// LS Electric XG5000 project: 2VFD2PUMPS
// PLC LSPLC

PROGRAM ECODELI (task: Scan Program)

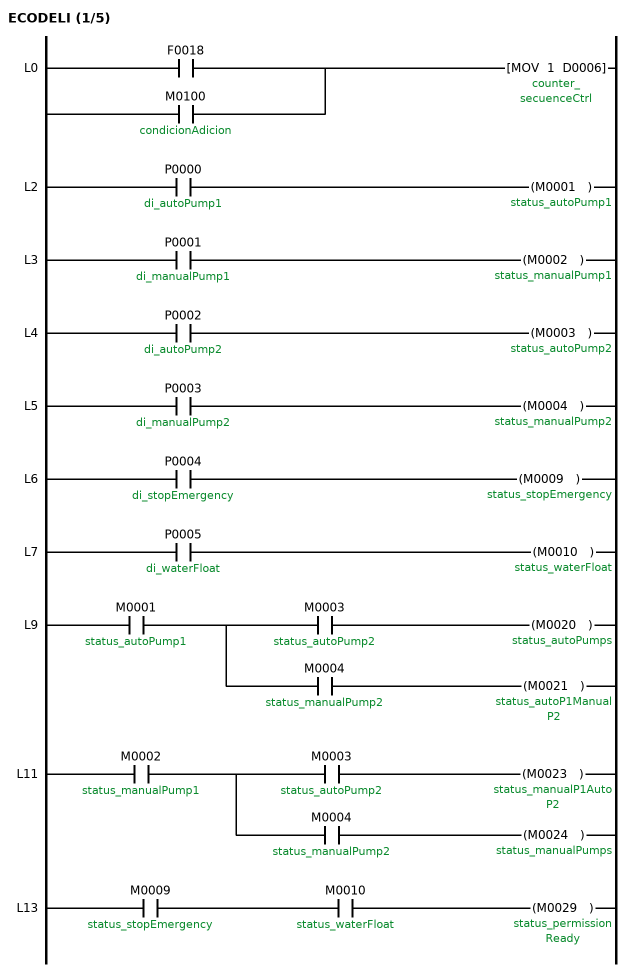
; L0
LOAD      F0018
OR        M0100	// condicionAdicion
MOV       1 D0006	// counter_secuenceCtrl
; L2
LOAD      P0000	// di_autoPump1
OUT       M0001	// status_autoPump1
; L3
LOAD      P0001	// di_manualPump1
OUT       M0002	// status_manualPump1
; L4
LOAD      P0002	// di_autoPump2
OUT       M0003	// status_autoPump2
; L5
LOAD      P0003	// di_manualPump2
OUT       M0004	// status_manualPump2
; L6
LOAD      P0004	// di_stopEmergency
OUT       M0009	// status_stopEmergency
; L7
LOAD      P0005	// di_waterFloat
OUT       M0010	// status_waterFloat
; L9
LOAD      M0001	// status_autoPump1
MPUSH
AND       M0003	// status_autoPump2
OUT       M0020	// status_autoPumps
MPOP
AND       M0004	// status_manualPump2
OUT       M0021	// status_autoP1ManualP2
; L11
LOAD      M0002	// status_manualPump1
MPUSH
AND       M0003	// status_autoPump2
OUT       M0023	// status_manualP1AutoP2
MPOP
AND       M0004	// status_manualPump2
OUT       M0024	// status_manualPumps
; L13
LOAD      M0009	// status_stopEmergency
AND       M0010	// status_waterFloat
OUT       M0029	// status_permissionReady

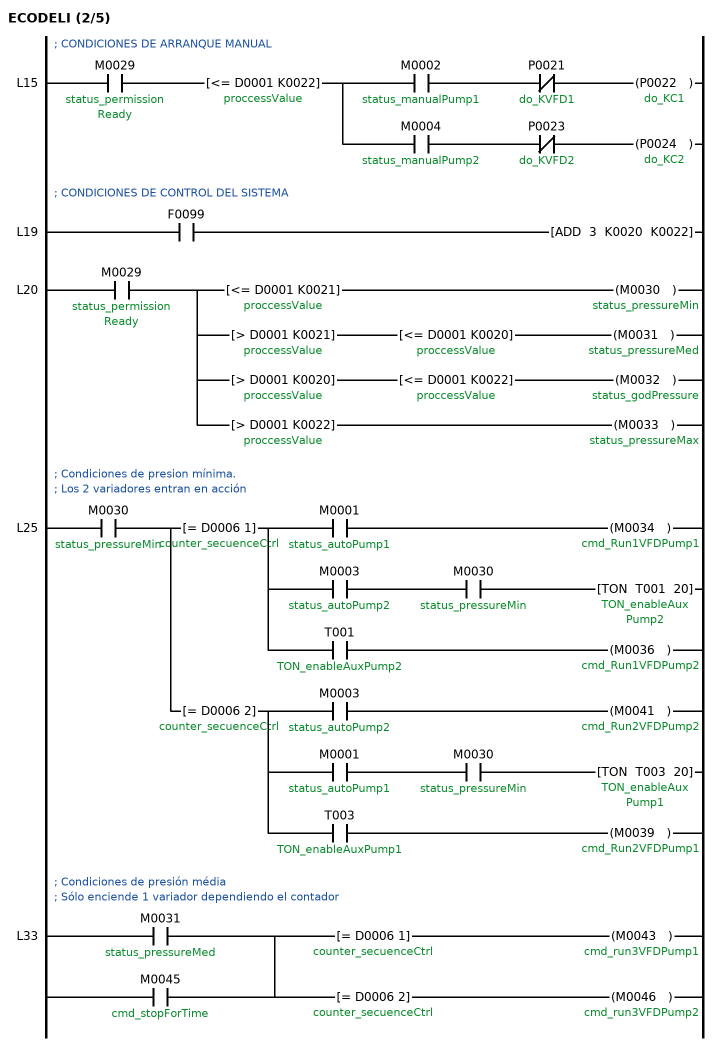
// CONDICIONES DE ARRANQUE MANUAL
; L15
LOAD      M0029	// status_permissionReady
AND<=     D0001 K0022	// proccessValue
MPUSH
AND       M0002	// status_manualPump1
AND NOT   P0021	// do_KVFD1
OUT       P0022	// do_KC1
MPOP
AND       M0004	// status_manualPump2
AND NOT   P0023	// do_KVFD2
OUT       P0024	// do_KC2
// CONDICIONES DE CONTROL DEL SISTEMA
; L19
LOAD      F0099
ADD       3 K0020 K0022
; L20
LOAD      M0029	// status_permissionReady
MPUSH
AND<=     D0001 K0021	// proccessValue
OUT       M0030	// status_pressureMin
MLOAD
AND>      D0001 K0021	// proccessValue
AND<=     D0001 K0020	// proccessValue
OUT       M0031	// status_pressureMed
MLOAD
AND>      D0001 K0020	// proccessValue
AND<=     D0001 K0022	// proccessValue
OUT       M0032	// status_godPressure
MPOP
AND>      D0001 K0022	// proccessValue
OUT       M0033	// status_pressureMax
// Condiciones de presion mínima.
// Los 2 variadores entran en acción
; L25
LOAD      M0030	// status_pressureMin
MPUSH
AND=      D0006 1	// counter_secuenceCtrl
MPUSH
AND       M0001	// status_autoPump1
OUT       M0034	// cmd_Run1VFDPump1
MLOAD
AND       M0003	// status_autoPump2
AND       M0030	// status_pressureMin
TON       T001 20	// TON_enableAuxPump2
MPOP
AND       T001	// TON_enableAuxPump2
OUT       M0036	// cmd_Run1VFDPump2
MPOP
AND=      D0006 2	// counter_secuenceCtrl
MPUSH
AND       M0003	// status_autoPump2
OUT       M0041	// cmd_Run2VFDPump2
MLOAD
AND       M0001	// status_autoPump1
AND       M0030	// status_pressureMin
TON       T003 20	// TON_enableAuxPump1
MPOP
AND       T003	// TON_enableAuxPump1
OUT       M0039	// cmd_Run2VFDPump1
// Condiciones de presión média
// Sólo enciende 1 variador dependiendo el contador
; L33
LOAD      M0031	// status_pressureMed
OR        M0045	// cmd_stopForTime
MPUSH
AND=      D0006 1	// counter_secuenceCtrl
OUT       M0043	// cmd_run3VFDPump1
MPOP
AND=      D0006 2	// counter_secuenceCtrl
OUT       M0046	// cmd_run3VFDPump2

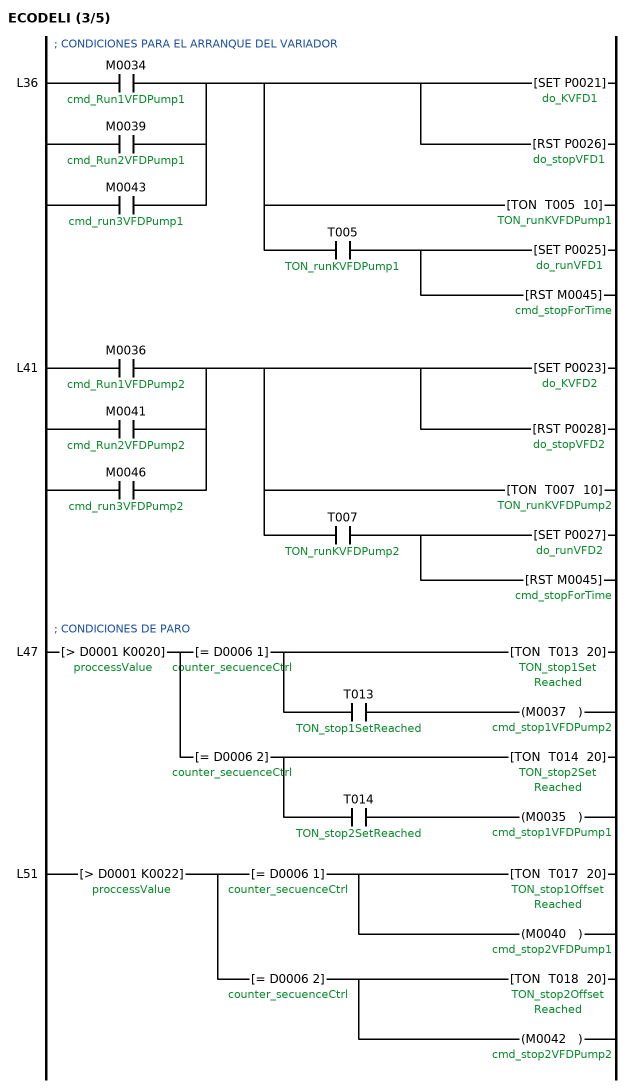
// CONDICIONES PARA EL ARRANQUE DEL VARIADOR
; L36
LOAD      M0034	// cmd_Run1VFDPump1
OR        M0039	// cmd_Run2VFDPump1
OR        M0043	// cmd_run3VFDPump1
SET       P0021	// do_KVFD1
RST       P0026	// do_stopVFD1
TON       T005 10	// TON_runKVFDPump1
AND       T005	// TON_runKVFDPump1
SET       P0025	// do_runVFD1
RST       M0045	// cmd_stopForTime
; L41
LOAD      M0036	// cmd_Run1VFDPump2
OR        M0041	// cmd_Run2VFDPump2
OR        M0046	// cmd_run3VFDPump2
SET       P0023	// do_KVFD2
RST       P0028	// do_stopVFD2
TON       T007 10	// TON_runKVFDPump2
AND       T007	// TON_runKVFDPump2
SET       P0027	// do_runVFD2
RST       M0045	// cmd_stopForTime
// CONDICIONES DE PARO
; L47
LOAD>     D0001 K0020	// proccessValue
MPUSH
AND=      D0006 1	// counter_secuenceCtrl
TON       T013 20	// TON_stop1SetReached
AND       T013	// TON_stop1SetReached
OUT       M0037	// cmd_stop1VFDPump2
MPOP
AND=      D0006 2	// counter_secuenceCtrl
TON       T014 20	// TON_stop2SetReached
AND       T014	// TON_stop2SetReached
OUT       M0035	// cmd_stop1VFDPump1
; L51
LOAD>     D0001 K0022	// proccessValue
MPUSH
AND=      D0006 1	// counter_secuenceCtrl
TON       T017 20	// TON_stop1OffsetReached
OUT       M0040	// cmd_stop2VFDPump1
MPOP
AND=      D0006 2	// counter_secuenceCtrl
TON       T018 20	// TON_stop2OffsetReached
OUT       M0042	// cmd_stop2VFDPump2

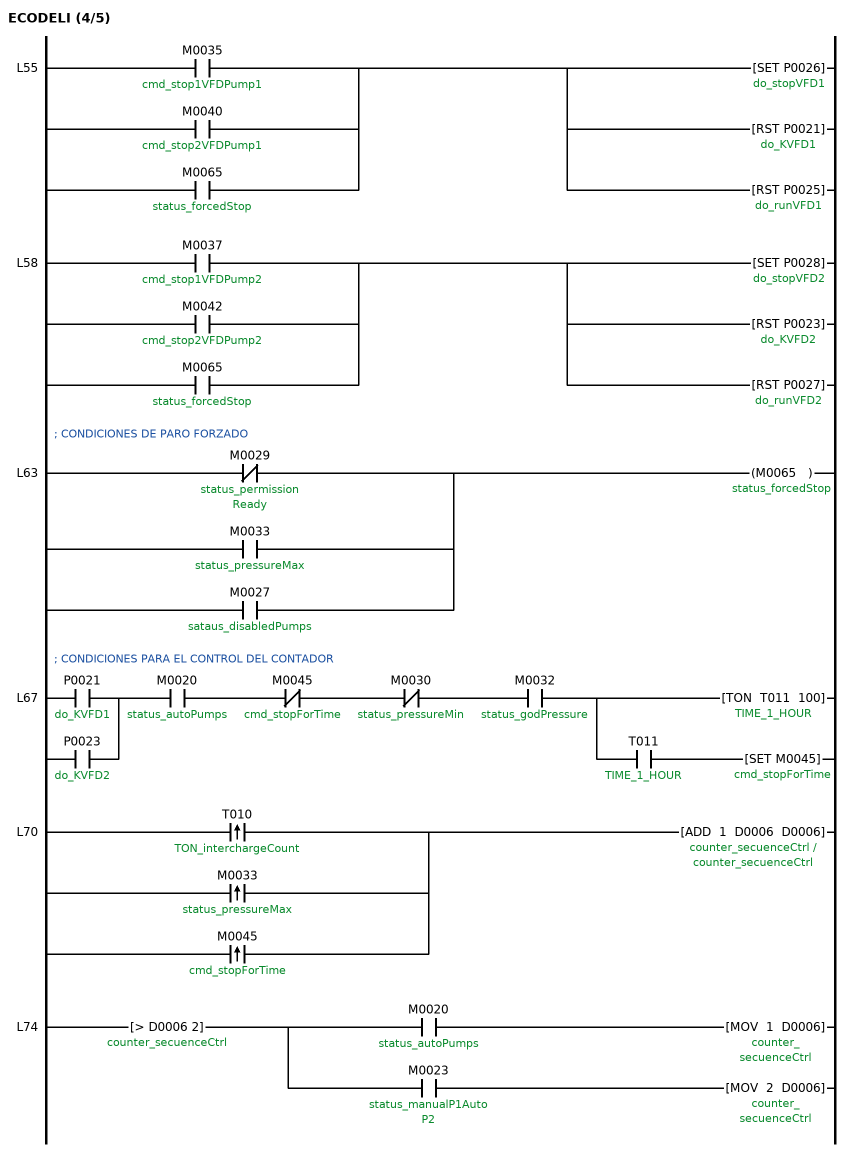
; L55
LOAD      M0035	// cmd_stop1VFDPump1
OR        M0040	// cmd_stop2VFDPump1
OR        M0065	// status_forcedStop
SET       P0026	// do_stopVFD1
RST       P0021	// do_KVFD1
RST       P0025	// do_runVFD1
; L58
LOAD      M0037	// cmd_stop1VFDPump2
OR        M0042	// cmd_stop2VFDPump2
OR        M0065	// status_forcedStop
SET       P0028	// do_stopVFD2
RST       P0023	// do_KVFD2
RST       P0027	// do_runVFD2
// CONDICIONES DE PARO FORZADO
; L63
LOAD NOT  M0029	// status_permissionReady
OR        M0033	// status_pressureMax
OR        M0027	// sataus_disabledPumps
OUT       M0065	// status_forcedStop
// CONDICIONES PARA EL CONTROL DEL CONTADOR
; L67
LOAD      P0021	// do_KVFD1
OR        P0023	// do_KVFD2
AND       M0020	// status_autoPumps
AND NOT   M0045	// cmd_stopForTime
AND NOT   M0030	// status_pressureMin
AND       M0032	// status_godPressure
TON       T011 100	// TIME_1_HOUR
AND       T011	// TIME_1_HOUR
SET       M0045	// cmd_stopForTime
; L70
LOADP     T010	// TON_interchargeCount
ORP       M0033	// status_pressureMax
ORP       M0045	// cmd_stopForTime
ADD       1 D0006 D0006	// counter_secuenceCtrl / counter_secuenceCtrl
; L74
LOAD>     D0006 2	// counter_secuenceCtrl
MPUSH
AND       M0020	// status_autoPumps
MOV       1 D0006	// counter_secuenceCtrl
MPOP
AND       M0023	// status_manualP1AutoP2
MOV       2 D0006	// counter_secuenceCtrl

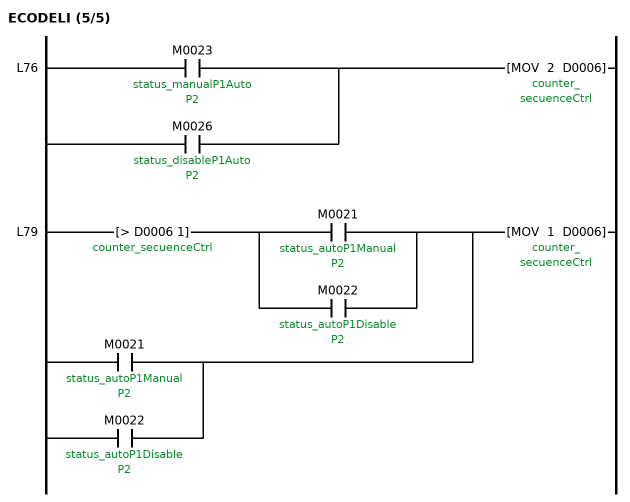
; L76
LOAD      M0023	// status_manualP1AutoP2
OR        M0026	// status_disableP1AutoP2
MOV       2 D0006	// counter_secuenceCtrl
; L79
LOAD>     D0006 1	// counter_secuenceCtrl
LOAD      M0021	// status_autoP1ManualP2
OR        M0022	// status_autoP1DisableP2
AND LOAD
OR        M0021	// status_autoP1ManualP2
OR        M0022	// status_autoP1DisableP2
MOV       1 D0006	// counter_secuenceCtrl

VARIABLES AND COMMENTS (devices not used above)
M00044	BIT	cmd_stop3VFDPump1
M00047	BIT	cmd_stop3VFDPump2
M00101	BIT	conditionstop2
M0255	WORD	contadoraux
M00050	BIT	interchangeForTime
M00051	BIT	interchanger2ForTime
K0023	WORD	MAX_PRESSURE
K0021	WORD	MIN_PRESSURE
M00110	BIT	nextCount
M00111	BIT	nextCount2
K0022	WORD	OFFSET_PRESSURE
K0020	WORD	SET_POINT
M00060	BIT	status_stopVFDPump1
M00061	BIT	status_stopVFDPump2
T0004	BIT/WORD	TON_disableAuxPump1
T0002	BIT/WORD	TON_disableAuxPump2
T0009	BIT/WORD	TON_interchargeForTime
T0015	BIT/WORD	TON_stop2KVFDPump1
T0016	BIT/WORD	TON_stop2KVFDPump2
T0006	BIT/WORD	TON_stopKVFDPump1
T0008	BIT/WORD	TON_stopKVFDPump2